FUNCTION F_STRING_TO_LINT : LINT
VAR_INPUT
	in_s:	STRING;
END_VAR
VAR
	lrVal:	LREAL;
END_VAR

// STRING_TO_LINT DOES NOT WORK !!!!!
//
// The string has to be converted to LREAL first and then to LINT
//
lrVal	:= STRING_TO_LREAL(in_s);

F_STRING_TO_LINT	:= LREAL_TO_LINT(lrVal);

END_FUNCTION

(* stored: Version 1.1.0.1, ProductVersion 3.1.4024.10
   POU F_STRING_TO_LINT: Id {b381afd4-c76e-4682-9efd-2bb6c70b6483}, SpecialFunc None *)
